Staubli VAL3: printScroll.pgx

program printScroll()
  local num i
  local num lX
  local num lY
begin
  //-----------------------------------------------------------------------
  //Header begin
  //Description of program
  //  Put the scrool on the right of the list menu.
  //
  //History
  //  Creation : 28-04-08 - f.Rob
  //Header end
  //-----------------------------------------------------------------------
  if size(sItems)>nListHeight
    //Find the percentage
    //Windows style
    //i=(size(sItems)-nListHeight+1)/(nFirst+1)
    // nokia style
    i=(size(sItems))/(nFirst+nView+1)
    lX=nTopX+nBottomX+1
    lY=roundUp((nListHeight)/i+nTopY)
    for i=nTopY+1 to nListHeight
      gotoxy(lX,i)
      if i==lY
        //
        put("■")
        //
      else
        put("│")
      endIf
    endFor
  endIf
end
